TYPE T_Ctrl_SIf_ICL:
STRUCT
	///configuration
	Cfg: T_Ctrl_SIf_ICL_Cfg;
	///parameter
	Par: T_Ctrl_SIf_ICL_Par;
	///current values
	Cur: T_Ctrl_SIf_ICL_Cur;
	///io input
	In: T_Ctrl_SIf_ICL_In;
	///io output
	///alarm number used in this controller
	Alm: ARRAY[1..5] OF T_Ctrl_Alm;
END_STRUCT
END_TYPE

(* stored: Version 1.1.0.1, ProductVersion 3.1.0.19
   DUT T_Ctrl_SIf_ICL: Id {181a255c-5a7e-4292-b63e-ecfb6a6273b5} *)
